# EPICS substitutions: Module_8_Alarms_Archiver_Autosave_and_Restore/1_Alarms/SecondAirCond/AirCondSysApp/Db/AirCondSys.substitutions
# Air Conditioning System substitutions file

file "db/dbAirCondSys.db" {
    { user = "ac", InsulCoeff = 0.02, HighTmp = 50, LowTmp = 20, PreSetTmp = 25, DeadBand = 1, InitPower = 0.4, MaxPower = 0.5 }
}
